SUBAPPLICATION Uebung_034a1_Q4_AX (* Numeric Value Input auf PWM Ausgang (Adapter Version) *)
  (* Standard: 61499-2; Description: Copyright (c) 2023 Meisterschulen am Ostbahnhof This program and the accompanying materials are made available under the terms of the Eclipse Public License 2.0 which is available at https://www.eclipse.org/legal/epl-2.0/ SPDX-License-Identifier: EPL-2.0 *)
  (* Version 1.0, 2026-04-20, Franz Höpfinger, Meisterschulen am Ostbahnhof, initial API and implementation (Adapter Version) *)
  PACKAGE Uebungen;
  IMPORT Uebungen::const::UT::PWM::DefaultPool_PWM::InputNumber_PWM_Value;
  IMPORT logiBUS::io::DQ::logiBUS_DO::Output_Q4;
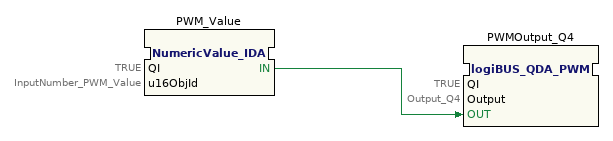
  (* ACHTUNG !! Ereignis erscheint erst im Adapter, wenn man die Numeric Value mit OK Bestätigt. nicht bei Button Druck. *)
  FBS
    PWMOutput_Q4 : logiBUS::io::DQ::logiBUS_QDA_PWM(QI := TRUE, Output := Output_Q4);
    PWM_Value : isobus::UT::io::NumericValue::NumericValue_IDA(QI := TRUE, u16ObjId := InputNumber_PWM_Value);
  END_FBS
  ADAPTER_CONNECTIONS
    PWM_Value.IN TO PWMOutput_Q4.OUT;
  END_CONNECTIONS
END_SUBAPPLICATION
